// TwinCAT 3 PLC project MiniRobotPLC
// ProgramVersion: 3.1.4024.0
// libraries:
//   CL_GreenhouseObjectsLibrary, * (CleanGreensSA)
//   Tc2_MC2, * (Beckhoff Automation GmbH)
//   Tc2_Standard, * (Beckhoff Automation GmbH)
//   Tc2_System, * (Beckhoff Automation GmbH)
//   Tc3_Module, * (Beckhoff Automation GmbH)
// project tree:
//   DUTs/ E_RequAxle.TcDUT, E_StepAxle.TcDUT, MainStm.TcDUT, ST_AnalogLimits.TcDUT, ST_Analog_HWI.TcDUT, ST_Axle.TcDUT, ST_CardState_HWI.TcDUT, ST_DriverAX8206_HWI.TcDUT, ST_GHMI.TcDUT, ST_HMI.TcDUT, ST_IrrigationLine.TcDUT, ST_JogMotorControl.TcDUT, ST_MainCabinet_HWI.TcDUT, ST_MainCabinet_HWQ.TcDUT, ST_MainPwrPhases_HWI.TcDUT, ST_ManualCtrlBtn.TcDUT, ST_OverCurrProtection_HWI.TcDUT, ST_OverCurrProtection_HWQ.TcDUT, ST_PhaseInfo.TcDUT, ST_PhasesCommon.TcDUT, ST_PositioningLaser_HWI.TcDUT, ST_PwrSupplyAX8620_HWI.TcDUT, ST_RemoteControl_HWI.TcDUT, ST_RobotIdentification_HWI.TcDUT, ST_RobotLineBox_HWI.TcDUT, ST_RobotLineBox_HWQ.TcDUT, ST_Robot_Axes.TcDUT, ST_Robot_HWI.TcDUT, ST_Robot_HWQ.TcDUT, ST_SystemStatus.TcDUT, ST_SystemStatus_AR.TcDUT, ST_SystemStatus_ARP.TcDUT, ST_UPS_HWI.TcDUT
//   GVLs/ G.TcGVL, GI.TcGVL (excluded from build), GIQ_Robot01.TcGVL, GQ.TcGVL
//   / PlcTask.TcTTO
//   POUs/ MAIN.TcPOU
// real-time tasks:
//   TASK PlcTask: cycle T#10ms, priority 20, ADS port 350
// motion (NC):
//   TASK NC-Task 1 SAF: cycle T#2ms, priority 4, ADS port 501
//   TASK NC-Task 1 SVB: cycle T#10ms, priority 8, ADS port 511
//   AXIS Axis 1 (id 1)
//     OtherSettings: AllowMotionCmdToSlave=true
//     encoder EncType=19
//       EncPara: MaxCount=#xffffffff
//     drive DrvType=16
//       DrvPara: MaxCount=#xffffffff, DriveControlDWord=#x00000100
//         Analog: TorqueSetpointScale=10, ScaleFactorActTorque=0.1
//         TimeComp: TaskDelayCycles=1
//     controller CtrType=1
//       CtrPara: PriorControlFactor=1
//         Observer: BandWidth=20
//   AXIS Axis 2 (id 2)
//     OtherSettings: AllowMotionCmdToSlave=true
//     encoder EncType=19
//       EncPara: MaxCount=#xffffffff
//     drive DrvType=16
//       DrvPara: MaxCount=#xffffffff, DriveControlDWord=#x00000100
//         Analog: TorqueSetpointScale=10, ScaleFactorActTorque=0.1
//         TimeComp: TaskDelayCycles=1
//     controller CtrType=1
//       CtrPara: PriorControlFactor=1
//         Observer: BandWidth=20
//   AXIS Axis 3 (id 3)
//     OtherSettings: AllowMotionCmdToSlave=true
//     encoder EncType=19
//       EncPara: MaxCount=#xffffffff
//     drive DrvType=16
//       DrvPara: MaxCount=#xffffffff, DriveControlDWord=#x00000100
//         Analog: TorqueSetpointScale=10, ScaleFactorActTorque=0.1
//         TimeComp: TaskDelayCycles=1
//     controller CtrType=1
//       CtrPara: PriorControlFactor=1
//         Observer: BandWidth=20
//   AXIS Axis 4 (id 4)
//     OtherSettings: AllowMotionCmdToSlave=true
//     encoder EncType=19
//       EncPara: MaxCount=#xffffffff
//     drive DrvType=16
//       DrvPara: MaxCount=#xffffffff, DriveControlDWord=#x00000100
//         Analog: TorqueSetpointScale=10, ScaleFactorActTorque=0.1
//         TimeComp: TaskDelayCycles=1
//     controller CtrType=1
//       CtrPara: PriorControlFactor=1
//         Observer: BandWidth=20
//   AXIS CGSMini_Robot01AxisLine1Front (id 5)
//     OtherSettings: AllowMotionCmdToSlave=true
//     encoder EncType=1
//     drive DrvType=5
//       Analog: TorqueSetpointScale=10, ScaleFactorActTorque=0.1
//     controller CtrType=1
//       CtrPara: PriorControlFactor=1
//         Observer: BandWidth=20
//   AXIS CGSMini_Robot01AxisLine1Back (id 6)
//     OtherSettings: AllowMotionCmdToSlave=true
//     encoder EncType=1
//     drive DrvType=5
//       Analog: TorqueSetpointScale=10, ScaleFactorActTorque=0.1
//     controller CtrType=1
//       CtrPara: PriorControlFactor=1
//         Observer: BandWidth=20
//   AXIS CGSMini_Robot01AxisLine2Front (id 7)
//     OtherSettings: AllowMotionCmdToSlave=true
//     encoder EncType=1
//     drive DrvType=5
//       Analog: TorqueSetpointScale=10, ScaleFactorActTorque=0.1
//     controller CtrType=1
//       CtrPara: PriorControlFactor=1
//         Observer: BandWidth=20
//   AXIS CGSMini_Robot01AxisLine2Back (id 8)
//     OtherSettings: AllowMotionCmdToSlave=true
//     encoder EncType=1
//     drive DrvType=5
//       Analog: TorqueSetpointScale=10, ScaleFactorActTorque=0.1
//     controller CtrType=1
//       CtrPara: PriorControlFactor=1
//         Observer: BandWidth=20
// I/O:
//   DEVICE CGSMini_IRSMainPLCNoSafe, AmsNetId 5.93.147.0.3.1
//     CGSMini_RobotAllMainCab-EL1200
// variable links:
//   MiniRobotPLC Instance <-> CGSMini_IRSMainPLCNoSafe/CGSMini_RobotAllMainCab-EL1200/CGSMini_Robot01LineBoxAnaInN01-EL3202
//     PlcTask Inputs/GIQ_Robot01.stBoxIN/stAnaInN01_3202State/uiDataState <-> InfoData/State
//     PlcTask Inputs/GIQ_Robot01.stBoxIN/stAnaRTDLine1/bTError <-> RTD1/Status/Error
//     PlcTask Inputs/GIQ_Robot01.stBoxIN/stAnaRTDLine2/bTError <-> RTD2/Status/Error
//     PlcTask Inputs/GIQ_Robot01.stBoxIN/stAnaRTDLine1/bTLimit1 <-> RTD1/Status/Limit 1
//     PlcTask Inputs/GIQ_Robot01.stBoxIN/stAnaRTDLine1/bTLimit2 <-> RTD1/Status/Limit 2
//     PlcTask Inputs/GIQ_Robot01.stBoxIN/stAnaRTDLine2/bTLimit1 <-> RTD2/Status/Limit 1
//     PlcTask Inputs/GIQ_Robot01.stBoxIN/stAnaRTDLine2/bTLimit2 <-> RTD2/Status/Limit 2
//     PlcTask Inputs/GIQ_Robot01.stBoxIN/stAnaRTDLine1/bTOverRange <-> RTD1/Status/Overrange
//     PlcTask Inputs/GIQ_Robot01.stBoxIN/stAnaRTDLine2/bTOverRange <-> RTD2/Status/Overrange
//     PlcTask Inputs/GIQ_Robot01.stBoxIN/stAnaRTDLine1/bTUnderRange <-> RTD1/Status/Underrange
//     PlcTask Inputs/GIQ_Robot01.stBoxIN/stAnaRTDLine2/bTUnderRange <-> RTD2/Status/Underrange
//     PlcTask Inputs/GIQ_Robot01.stBoxIN/stAnaRTDLine1/siAnaRaw <-> RTD1/Value
//     PlcTask Inputs/GIQ_Robot01.stBoxIN/stAnaRTDLine2/siAnaRaw <-> RTD2/Value
//   MiniRobotPLC Instance <-> CGSMini_IRSMainPLCNoSafe/CGSMini_RobotAllMainCab-EL1200/CGSMini_Robot01LineBoxAnaInN02-EL3054
//     PlcTask Inputs/GIQ_Robot01.stBoxIN/stAnaFlowLine1/bTError <-> Flow1/Status/Error
//     PlcTask Inputs/GIQ_Robot01.stBoxIN/stAnaFlowLine2/bTError <-> Flow2/Status/Error
//     PlcTask Inputs/GIQ_Robot01.stBoxIN/stAnaFlowLine1/bTLimit1 <-> Flow1/Status/Limit 1
//     PlcTask Inputs/GIQ_Robot01.stBoxIN/stAnaFlowLine1/bTLimit2 <-> Flow1/Status/Limit 2
//     PlcTask Inputs/GIQ_Robot01.stBoxIN/stAnaFlowLine2/bTLimit1 <-> Flow2/Status/Limit 1
//     PlcTask Inputs/GIQ_Robot01.stBoxIN/stAnaFlowLine2/bTLimit2 <-> Flow2/Status/Limit 2
//     PlcTask Inputs/GIQ_Robot01.stBoxIN/stAnaFlowLine1/bTOverRange <-> Flow1/Status/Overrange
//     PlcTask Inputs/GIQ_Robot01.stBoxIN/stAnaFlowLine2/bTOverRange <-> Flow2/Status/Overrange
//     PlcTask Inputs/GIQ_Robot01.stBoxIN/stAnaFlowLine1/bTUnderRange <-> Flow1/Status/Underrange
//     PlcTask Inputs/GIQ_Robot01.stBoxIN/stAnaFlowLine2/bTUnderRange <-> Flow2/Status/Underrange
//     PlcTask Inputs/GIQ_Robot01.stBoxIN/stAnaFlowLine1/siAnaRaw <-> Flow1/Value
//     PlcTask Inputs/GIQ_Robot01.stBoxIN/stAnaFlowLine2/siAnaRaw <-> Flow2/Value
//     PlcTask Inputs/GIQ_Robot01.stBoxIN/stAnaInN02_3054State/uiDataState <-> InfoData/State
//     PlcTask Inputs/GIQ_Robot01.stBoxIN/stAnaPressure/bTError <-> Pressure1/Status/Error
//     PlcTask Inputs/GIQ_Robot01.stBoxIN/stAnaPressure/bTLimit1 <-> Pressure1/Status/Limit 1
//     PlcTask Inputs/GIQ_Robot01.stBoxIN/stAnaPressure/bTLimit2 <-> Pressure1/Status/Limit 2
//     PlcTask Inputs/GIQ_Robot01.stBoxIN/stAnaPressure/bTOverRange <-> Pressure1/Status/Overrange
//     PlcTask Inputs/GIQ_Robot01.stBoxIN/stAnaPressure/bTUnderRange <-> Pressure1/Status/Underrange
//     PlcTask Inputs/GIQ_Robot01.stBoxIN/stAnaPressure/siAnaRaw <-> Pressure1/Value
//   MiniRobotPLC Instance <-> CGSMini_IRSMainPLCNoSafe/CGSMini_RobotAllMainCab-EL1200/CGSMini_Robot01LineBoxAnaInN03-EL3202
//     PlcTask Inputs/GIQ_Robot01.stBoxIN/stAnaInN03_3202State/uiDataState <-> InfoData/State
//     PlcTask Inputs/GIQ_Robot01.stBoxIN/stAnaRTDExternal/bTError <-> RTDExternal/Status/Error
//     PlcTask Inputs/GIQ_Robot01.stBoxIN/stAnaRTDExternal/bTLimit1 <-> RTDExternal/Status/Limit 1
//     PlcTask Inputs/GIQ_Robot01.stBoxIN/stAnaRTDExternal/bTLimit2 <-> RTDExternal/Status/Limit 2
//     PlcTask Inputs/GIQ_Robot01.stBoxIN/stAnaRTDExternal/bTOverRange <-> RTDExternal/Status/Overrange
//     PlcTask Inputs/GIQ_Robot01.stBoxIN/stAnaRTDExternal/bTUnderRange <-> RTDExternal/Status/Underrange
//     PlcTask Inputs/GIQ_Robot01.stBoxIN/stAnaRTDExternal/siAnaRaw <-> RTDExternal/Value
//     PlcTask Inputs/GIQ_Robot01.stBoxIN/stAnaRTDInternal/bTError <-> RTDInternal/Status/Error
//     PlcTask Inputs/GIQ_Robot01.stBoxIN/stAnaRTDInternal/bTLimit1 <-> RTDInternal/Status/Limit 1
//     PlcTask Inputs/GIQ_Robot01.stBoxIN/stAnaRTDInternal/bTLimit2 <-> RTDInternal/Status/Limit 2
//     PlcTask Inputs/GIQ_Robot01.stBoxIN/stAnaRTDInternal/bTOverRange <-> RTDInternal/Status/Overrange
//     PlcTask Inputs/GIQ_Robot01.stBoxIN/stAnaRTDInternal/bTUnderRange <-> RTDInternal/Status/Underrange
//     PlcTask Inputs/GIQ_Robot01.stBoxIN/stAnaRTDInternal/siAnaRaw <-> RTDInternal/Value
//   MiniRobotPLC Instance <-> CGSMini_IRSMainPLCNoSafe/CGSMini_RobotAllMainCab-EL1200/CGSMini_Robot01LineBoxInN01-EL1008
//     PlcTask Inputs/GIQ_Robot01.stBoxIN/stInN01_1008State/uiDataState <-> InfoData/State
//     PlcTask Inputs/GIQ_Robot01.stBoxIN/stRemoteCtrl/BtnBackwardMan <-> Channel 2/BtnBackwardMan
//     PlcTask Inputs/GIQ_Robot01.stBoxIN/stRemoteCtrl/BtnForwardMan <-> Channel 1/BtnForwardMan
//     PlcTask Inputs/GIQ_Robot01.stBoxIN/stRemoteCtrl/BtnValveLine1Man <-> Channel 3/BtnValveLine1Man
//     PlcTask Inputs/GIQ_Robot01.stBoxIN/stRemoteCtrl/BtnValveLine2Man <-> Channel 4/BtnValveLine2Man
//     PlcTask Inputs/GIQ_Robot01.stBoxIN/stRobotID/bSelBit0 <-> Channel 5/SelLineBit0
//     PlcTask Inputs/GIQ_Robot01.stBoxIN/stRobotID/bSelBit1 <-> Channel 6/SelLineBit1
//     PlcTask Inputs/GIQ_Robot01.stBoxIN/stRobotID/bSelBit2 <-> Channel 7/SelLineBit2
//     PlcTask Inputs/GIQ_Robot01.stBoxIN/stRobotID/bSelBit3 <-> Channel 8/SelLineBit3
//   MiniRobotPLC Instance <-> CGSMini_IRSMainPLCNoSafe/CGSMini_RobotAllMainCab-EL1200/CGSMini_Robot01LineBoxOverCurrProt1-EL9222
//     PlcTask Inputs/GIQ_Robot01.stBoxIN/stOverCProt1_9222State/uiDataState <-> InfoData/State
//     PlcTask Inputs/GIQ_Robot01.stBoxIN/stOverCProt/bEnabled <-> OCP Inputs Channel 1/Status/Enabled
//     PlcTask Inputs/GIQ_Robot01.stBoxIN/stOverCProt/bError <-> OCP Inputs Channel 1/Status/Error
//   MiniRobotPLC Instance <-> CGSMini_IRSMainPLCNoSafe/CGSMini_RobotAllMainCab-EL1200/CGSMini_Robot01MainCabEtherCATBusEK1122/CGSMini_Robot01Laser-SickDL100
//     PlcTask Inputs/GIQ_Robot01.stIN/stLaserPos <-> Distance/Distance
//     PlcTask Inputs/GIQ_Robot01.stIN/stLaserPos_State/uiDataState <-> InfoData/State
//   MiniRobotPLC Instance <-> CGSMini_IRSMainPLCNoSafe/CGSMini_RobotAllMainCab-EL1200/CGSMini_Robot01MainCabEtherCATBusEK1122/CGSMini_Robot01OnboardAxisPwrSupply-AX8620
//     PlcTask Inputs/GIQ_Robot01.stIN/stPwrSupplyAX8620/bFanMalfunc <-> PSM Warning register/Warning/A4 Fan malfunction
//     PlcTask Inputs/GIQ_Robot01.stIN/stPwrSupplyAX8620/bOverTemp <-> PSM Warning register/Warning/A2 Device overtemperature
//     PlcTask Inputs/GIQ_Robot01.stIN/stPwrSupplyAX8620/bOverVoltage <-> PSM Warning register/Warning/A5 Mains overvoltage
//     PlcTask Inputs/GIQ_Robot01.stIN/stPwrSupplyAX8620/bUnderVoltage <-> PSM Warning register/Warning/A6 Mains undervoltage
//     PlcTask Inputs/GIQ_Robot01.stIN/stPwrSupplyAX8620/comState/bWcState <-> WcState/WcState
//     PlcTask Inputs/GIQ_Robot01.stIN/stPwrSupplyAX8620/comState/uiDataState <-> InfoData/State
//     PlcTask Inputs/GIQ_Robot01.stIN/stPwrSupplyAX8620/sdiDcInputShift <-> InfoData/DcInputShift
//     PlcTask Inputs/GIQ_Robot01.stIN/stPwrSupplyAX8620/sdiDcOutputShift <-> InfoData/DcOutputShift
//   MiniRobotPLC Instance <-> CGSMini_IRSMainPLCNoSafe/CGSMini_RobotAllMainCab-EL1200/CGSMini_Robot01MainCabEtherCATBusEK1122/CGSMini_Robot01OnboardAxisPwrSupply-AX8620/CGSMini_Robot01OnboardAxisDriverLine1-AX8206
//     PlcTask Inputs/GIQ_Robot01.stIN/stDriverLine1/comState <-> InfoData/State
//     PlcTask Inputs/GIQ_Robot01.stIN/stDriverLine1/rBackMotorTemp <-> Back/Ch A SyncServoMotor Inputs/Actual motor temperature
//     PlcTask Inputs/GIQ_Robot01.stIN/stDriverLine1/rBackMotorTorque <-> Back/Ch A TorqueControl Inputs/Ch A Torque/force actual value
//     PlcTask Inputs/GIQ_Robot01.stIN/stDriverLine1/rFrontMotorTemp <-> Front/Ch B SyncServoMotor Inputs/Actual motor temperature
//     PlcTask Inputs/GIQ_Robot01.stIN/stDriverLine1/rFrontMotorTorque <-> Front/Ch B TorqueControl Inputs/Ch B Torque/force actual value
//     PlcTask Inputs/GIQ_Robot01.stIN/stDriverLine1/sdiDcInputShift <-> InfoData/DcInputShift
//     PlcTask Inputs/GIQ_Robot01.stIN/stDriverLine1/sdiDcOutputShift <-> InfoData/DcOutputShift
//     PlcTask Inputs/GIQ_Robot01.stIN/stDriverLine1/siBackIGBTTemp <-> Back/Ch A AxisMain Inputs/IGBT temperature
//     PlcTask Inputs/GIQ_Robot01.stIN/stDriverLine1/siFrontIGBTTemp <-> Front/Ch B AxisMain Inputs/IGBT temperature
//     PlcTask Inputs/GIQ_Robot01.stIN/stDriverLine1/udBackMotorDIGIns <-> Back/Ch A AxisMain Inputs/Ch A Digital inputs
//     PlcTask Inputs/GIQ_Robot01.stIN/stDriverLine1/udFrontMotorDIGIns <-> Front/Ch B AxisMain Inputs/Ch B Digital inputs
//   MiniRobotPLC Instance <-> CGSMini_IRSMainPLCNoSafe/CGSMini_RobotAllMainCab-EL1200/CGSMini_Robot01MainCabEtherCATBusEK1122/CGSMini_Robot01OnboardAxisPwrSupply-AX8620/CGSMini_Robot01OnboardAxisDriverLine2-AX8206
//     PlcTask Inputs/GIQ_Robot01.stIN/stDriverLine2/comState <-> InfoData/State
//     PlcTask Inputs/GIQ_Robot01.stIN/stDriverLine2/rBackMotorTemp <-> Back/Ch A SyncServoMotor Inputs/Actual motor temperature
//     PlcTask Inputs/GIQ_Robot01.stIN/stDriverLine2/rBackMotorTorque <-> Back/Ch A TorqueControl Inputs/Ch A Torque/force actual value
//     PlcTask Inputs/GIQ_Robot01.stIN/stDriverLine2/rFrontMotorTemp <-> Front/Ch B SyncServoMotor Inputs/Actual motor temperature
//     PlcTask Inputs/GIQ_Robot01.stIN/stDriverLine2/rFrontMotorTorque <-> Front/Ch B TorqueControl Inputs/Ch B Torque/force actual value
//     PlcTask Inputs/GIQ_Robot01.stIN/stDriverLine2/sdiDcInputShift <-> InfoData/DcInputShift
//     PlcTask Inputs/GIQ_Robot01.stIN/stDriverLine2/sdiDcOutputShift <-> InfoData/DcOutputShift
//     PlcTask Inputs/GIQ_Robot01.stIN/stDriverLine2/siBackIGBTTemp <-> Back/Ch A AxisMain Inputs/IGBT temperature
//     PlcTask Inputs/GIQ_Robot01.stIN/stDriverLine2/siFrontIGBTTemp <-> Front/Ch B AxisMain Inputs/IGBT temperature
//     PlcTask Inputs/GIQ_Robot01.stIN/stDriverLine2/udBackMotorDIGIns <-> Back/Ch A AxisMain Inputs/Ch A Digital inputs
//     PlcTask Inputs/GIQ_Robot01.stIN/stDriverLine2/udFrontMotorDIGIns <-> Front/Ch B AxisMain Inputs/Ch B Digital inputs
//   MiniRobotPLC Instance <-> CGSMini_IRSMainPLCNoSafe/CGSMini_RobotAllMainCab-EL1200/CGSMini_Robot01MainCabEtherCATBusEK1122/CGSMini_Robot01OnboardBox-EK1100
//     PlcTask Inputs/GIQ_Robot01.stIN/stOnboardBox_1100State/uiDataState <-> InfoData/State
//   MiniRobotPLC Instance <-> CGSMini_IRSMainPLCNoSafe/CGSMini_RobotAllMainCab-EL1200/CGSMini_Robot01MainCabEtherCATBusEK1122/CGSMini_Robot01OnboardBox-EK1100/CGSMini_Robot01OnBoardBoxAnaInN04-EL3054
//     PlcTask Inputs/GIQ_Robot01.stIN/stAnaInN04_3054State/uiDataState <-> InfoData/State
//     PlcTask Inputs/GIQ_Robot01.stIN/stAnaOnboardSpare1/bTError <-> Spare1/Status/Error
//     PlcTask Inputs/GIQ_Robot01.stIN/stAnaOnboardSpare1/bTLimit1 <-> Spare1/Status/Limit 1
//     PlcTask Inputs/GIQ_Robot01.stIN/stAnaOnboardSpare1/bTLimit2 <-> Spare1/Status/Limit 2
//     PlcTask Inputs/GIQ_Robot01.stIN/stAnaOnboardSpare1/bTOverRange <-> Spare1/Status/Overrange
//     PlcTask Inputs/GIQ_Robot01.stIN/stAnaOnboardSpare1/bTUnderRange <-> Spare1/Status/Underrange
//     PlcTask Inputs/GIQ_Robot01.stIN/stAnaOnboardSpare1/siAnaRaw <-> Spare1/Value
//   MiniRobotPLC Instance <-> CGSMini_IRSMainPLCNoSafe/CGSMini_RobotAllMainCab-EL1200/CGSMini_Robot01MainCabEtherCATBusEK1122/CGSMini_Robot01OnboardBox-EK1100/CGSMini_Robot01OnBoardBoxOutN01-EL2008
//     PlcTask Inputs/GIQ_Robot01.stIN/stOutN01_2008State/uiDataState <-> InfoData/State
//     PlcTask Outputs/G.outTest14 <-> Channel 8/Output
//     PlcTask Outputs/GIQ_Robot01.stOUT/FlushFloor <-> Channel 1/FlushFloor
//     PlcTask Outputs/GIQ_Robot01.stOUT/IrrigLine1 <-> Channel 3/IrrigLine1
//     PlcTask Outputs/GIQ_Robot01.stOUT/IrrigLine2 <-> Channel 4/IrrigLine2
//   MiniRobotPLC Instance <-> CGSMini_IRSMainPLCNoSafe/CGSMini_RobotAllMainCab-EL1200/CGSMini_RobotAllMainCabOutN01-EL2008
//     PlcTask Outputs/GQ.stMainCabinet/bEmgyBtnRedLight <-> Channel 3/EmgyBtnRedLight
//     PlcTask Outputs/GQ.stMainCabinet/bEmgyBtnWhiteLight <-> Channel 2/EmgyBtnWhiteLight
//     PlcTask Outputs/GQ.stMainCabinet/stStackLight/bBlue <-> Channel 4/blue
//     PlcTask Outputs/GQ.stMainCabinet/stStackLight/bBuzzer <-> Channel 8/buzzer
//     PlcTask Outputs/GQ.stMainCabinet/stStackLight/bGreen <-> Channel 5/green
//     PlcTask Outputs/GQ.stMainCabinet/stStackLight/bOrange <-> Channel 6/orange
//     PlcTask Outputs/GQ.stMainCabinet/stStackLight/bRed <-> Channel 7/red
//   MiniRobotPLC Instance <-> NC-Task 1 SAF/Axes/CGSMini_Robot01AxisLine1Back
//     PlcTask Inputs/GIQ_Robot01.stAxes.Line1Back.NcToPlc <-> Outputs/ToPlc
//     PlcTask Outputs/GIQ_Robot01.stAxes.Line1Back.PlcToNc <-> Inputs/FromPlc
//   MiniRobotPLC Instance <-> NC-Task 1 SAF/Axes/CGSMini_Robot01AxisLine1Front
//     PlcTask Inputs/GIQ_Robot01.stAxes.Line1Front.NcToPlc <-> Outputs/ToPlc
//     PlcTask Outputs/GIQ_Robot01.stAxes.Line1Front.PlcToNc <-> Inputs/FromPlc
//   MiniRobotPLC Instance <-> NC-Task 1 SAF/Axes/CGSMini_Robot01AxisLine2Back
//     PlcTask Inputs/GIQ_Robot01.stAxes.Line2Back.NcToPlc <-> Outputs/ToPlc
//     PlcTask Outputs/GIQ_Robot01.stAxes.Line2Back.PlcToNc <-> Inputs/FromPlc
//   MiniRobotPLC Instance <-> NC-Task 1 SAF/Axes/CGSMini_Robot01AxisLine2Front
//     PlcTask Inputs/GIQ_Robot01.stAxes.Line2Front.NcToPlc <-> Outputs/ToPlc
//     PlcTask Outputs/GIQ_Robot01.stAxes.Line2Front.PlcToNc <-> Inputs/FromPlc

CONFIGURATION MiniRobotPLC
    RESOURCE PLC ON TwinCAT3
        TASK PlcTask(INTERVAL := T#10ms, PRIORITY := 20);
        PROGRAM MAIN WITH PlcTask : MAIN;
    END_RESOURCE
END_CONFIGURATION

// ---- DUTs/E_RequAxle.TcDUT
{attribute 'qualified_only'}
{attribute 'strict'}
TYPE E_RequAxle :
(
  NoRequ := 0,
  PowerOn := 1,
  PowerOff := 2,
  Reset := 3,
  Jog := 4,
  Error := 254,
  Idle := 255
);
END_TYPE

// ---- DUTs/E_StepAxle.TcDUT
{attribute 'qualified_only'}
{attribute 'strict'}
TYPE E_StepAxle :
(
	//Idle	        := 0,
  Init          := 1,
  
	// STEPS ABSOLUTE
 	MoveAbs		    := 11,
	EndMoveAbs    := 12,
  
	// STEPS STOP
  InitStop      := 50,
	Stopping		  := 51,
  EndStopping   := 52,
	
	// STEPS HOMING
  InitHoming    := 60,
	Homing			  := 61,
  EndHoming     := 62,
  InitAbortHoming := 63,
  AbortHoming   := 64,
  InitRetryHoming := 65,
  RetryHoming     := 66,
	
	// STEPS Reset
  ResetTimeout := 70,
	Resetting	:= 71,
  ResetEnd := 72,
  
  // step jogs
  JogMoveFW := 80,
  JogMoveBW := 81,
  JogStop := 82,
  JogEnd := 83
);
END_TYPE

// ---- DUTs/MainStm.TcDUT
{attribute 'qualified_only'}
{attribute 'strict'}
TYPE MainStm :
(
	ModuleDatabaseInit := 0,
  ModuleDatabaseLoad,
  ErrorDatabaseInit,
	LoadSQLDB,
  Init,
	//WaitInitWebVISUTask,
	LoadModuleDB,
	InitWebVISUTask,
	IRSystemExec,//GreenhouseExec,
	PowerFailure,
	WaitPowerDown,
	ReqShutdown,
  ReqRestart,
  FailedLoadSQL,
  FailedInitObjects,
	End
);
END_TYPE

// ---- DUTs/ST_AnalogLimits.TcDUT
TYPE ST_AnalogLimits :
STRUCT
  lrAroundZero        : LREAL; //to check if the value is around zero
	lrRawLowerLimit		  : LREAL; // Lower limit for raw data
	lrRawUpperLimit		  : LREAL; // Upper limit for raw data
	lrScaleLowerLimit	  : LREAL; // Lower limit of scaled measurement
	lrScaleUpperLimit	  : LREAL; // Upper limit of scaled measurement
  bForceZero          : BOOL;
END_STRUCT
END_TYPE

// ---- DUTs/ST_Analog_HWI.TcDUT
TYPE ST_Analog_HWI :
STRUCT
  bTUnderRange      : BOOL;
  bTOverRange       : BOOL;
  bTLimit1          : BOOL;
  bTLimit2          : BOOL;
  bTError           : BOOL;
  siAnaRaw          : INT;  
END_STRUCT
END_TYPE

// ---- DUTs/ST_Axle.TcDUT
//Add Library Tc2_MC2
TYPE ST_Axle:
STRUCT
	stAxisRef						      : POINTER TO AXIS_REF;//axis reference linked to I/O
	fbPower						        : MC_Power;//Axis function - Power
	fbReset						        : MC_Reset;//Axis function - Reset
	fbSetPosition					    : MC_SetPosition;//Axis function - Set Position
	fbStop							      : MC_Stop;//stop
	fbHalt							      : MC_Halt;//Halt
	fbHome							      : MC_Home;//Home
	fbMoveJog							    : MC_Jog;//Jog
  fbReadStatus              : MC_ReadStatus;
	fbMoveAbsolute1				    : MC_MoveAbsolute;//	MC_MoveAbsolute1
  fbMoveAbsoluteWheelCheck  : MC_MoveAbsolute;// Add CustomAutomation 07.03.2023: Check du diamètre des roues 
  fbMoveAbsoluteCorrection  : MC_MoveAbsolute;// Add CustomAutomation 07.03.2023: Correction fin de parcours
 	fbMoveRelative					  : MC_MoveRelative;//Move Relative
	fbMoveVelocity					  : MC_MoveVelocity;//Move Velocity
	fbReadAxisError				    : MC_ReadAxisError;//Status and parameter - Read Axis Error
	fbReadActualPosition			: MC_ReadActualPosition;//Status and parameter - Read Actual Position
	fbReadActualVelocity			: MC_ReadActualVelocity;//Status and parameter - Read Actual Velocity
	fbGearInDyn					      : MC_GearInDyn;//Axis coupling - GearInDyn
	fbGearOut						      : MC_GearOut;//Axis coupling - GearOut
	fbPosCorrectionLimiter    : MC_PositionCorrectionLimiter;//Special extensions - Position Correction Limiter
	
	bGearOutDone					    : BOOL;
	bGearInDynDone					  : BOOL;
	bStopDone						      : BOOL;
END_STRUCT
END_TYPE

// ---- DUTs/ST_CardState_HWI.TcDUT
TYPE ST_CardState_HWI :
STRUCT
  uiDataState   : UINT;
  bWcState      : BOOL := FALSE;
END_STRUCT
END_TYPE

// ---- DUTs/ST_DriverAX8206_HWI.TcDUT

TYPE ST_DriverAX8206_HWI :
STRUCT
  comState          : ST_CardState_HWI;
  sdiDcOutputShift  : DINT;
  sdiDcInputShift   : DINT;

  siFrontIGBTTemp   : INT;//ChB
  siBackIGBTTemp    : INT;//ChA
  
  rFrontMotorTemp  : REAL;//ChB
  rBackMotorTemp   : REAL;//ChA
  
  rFrontMotorTorque : REAL;//ChB
  rBackMotorTorque  : REAL;//ChA
  
  udFrontMotorDIGIns: UDINT;//ChB
  udBackMotorDIGIns: UDINT;//ChA
END_STRUCT
END_TYPE

// ---- DUTs/ST_GHMI.TcDUT
TYPE ST_GHMI :
STRUCT
  bStartButton      		  : BOOL;
  bStopButton       		  : BOOL;
  bResetButton      		  : BOOL;
  bAbortButton      		  : BOOL;
  bClearButton      		  : BOOL;
  nIndexFrame       		  : INT := 0;
  nIndexFrameAdmin        : INT := 0;
  nIndexFrameHome   		  : INT := 0;
  bPopUpModulPresent		  : BOOL;
  bPopUpHoming      		  : BOOL;
  bPopUpExtractorAborted  : BOOL;
	bPopUpInsertModulesLine	: BOOL;
  bRestart          		  : BOOL;
  bShutdown          		  : BOOL;
	sBtnAdmin								: STRING(32);
END_STRUCT
END_TYPE

// ---- DUTs/ST_HMI.TcDUT
TYPE ST_HMI :
STRUCT
  nIrrLineSel  : UINT := 1;//at leat 1 robot line
END_STRUCT
END_TYPE

// ---- DUTs/ST_IrrigationLine.TcDUT
TYPE ST_IrrigationLine :
STRUCT
  stRobotLineBoxHWI   : POINTER TO ST_RobotLineBox_HWI;
  stRobotLineBoxHWQ   : POINTER TO ST_RobotLineBox_HWQ;
  stRobotHWI	        : POINTER TO ST_Robot_HWI;
  stRobotHWQ	        : POINTER TO ST_Robot_HWQ;
  stRobotAxes	        : POINTER TO ST_Robot_Axes;
END_STRUCT
END_TYPE

// ---- DUTs/ST_JogMotorControl.TcDUT
TYPE ST_JogMotorControl :
STRUCT
  bMoveFW   : BOOL := false;
  bMoveBW   : BOOL := false;
END_STRUCT
END_TYPE

// ---- DUTs/ST_MainCabinet_HWI.TcDUT
TYPE ST_MainCabinet_HWI :
STRUCT		
    //State
    stInN01_1008State       : ST_CardState_HWI;
    stOutN01_2008State      : ST_CardState_HWI; 
    stLicense_6070State     : ST_CardState_HWI; 
    stAnaInN01_3443         : ST_CardState_HWI; //CGSMini_RobotAllMainCabAnaInN01-EL3443
    
    //EK1122 ethercat State    
    stMainEK1122State       : ST_CardState_HWI;
    
		//inputs
		bKeyRestart			 	 			: BOOL;  
		bEmgyBtnCntct1					: BOOL; 
		bEmgyBtnCntct2	   			: BOOL;  
		bOverTemp45C			 			: BOOL := FALSE;  
    bPLCCircuitBreakerOpen  : BOOL := FALSE;   
    
    stUPS                   : ST_UPS_HWI;
    stPwrInfo               : ST_MainPwrPhases_HWI;
END_STRUCT
END_TYPE

// ---- DUTs/ST_MainCabinet_HWQ.TcDUT
TYPE ST_MainCabinet_HWQ :
STRUCT
  //outputs
  bEmgyBtnWhiteLight  	: BOOL;  
  bEmgyBtnRedLight  		: BOOL; 
  
  stStackLight          : ST_StackLight_HWQ;
END_STRUCT
END_TYPE

// ---- DUTs/ST_MainPwrPhases_HWI.TcDUT
TYPE ST_MainPwrPhases_HWI :
STRUCT
  L1 : ST_PhaseInfo;
  L2 : ST_PhaseInfo;
  L3 : ST_PhaseInfo;
  Tot : ST_PhasesCommon;
END_STRUCT
END_TYPE

// ---- DUTs/ST_ManualCtrlBtn.TcDUT
TYPE ST_ManualCtrlBtn :
STRUCT
  bMoveBackwardBtn        : BOOL := FALSE;
  bMoveForwardBtn         : BOOL := FALSE;
  bVlvLine1Btn            : BOOL := FALSE;
  bVlvLine2Btn            : BOOL := FALSE;
  
  bMoveBackwardBtnPress   : BOOL := FALSE;
  bMoveForwardBtnPress    : BOOL := FALSE;
  bVlvLine1BtnPress       : BOOL := FALSE;
  bVlvLine2BtnPress       : BOOL := FALSE;
END_STRUCT
END_TYPE

// ---- DUTs/ST_OverCurrProtection_HWI.TcDUT
TYPE ST_OverCurrProtection_HWI :
STRUCT
  bEnabled  : BOOL;
  bError    : BOOL;
END_STRUCT
END_TYPE

// ---- DUTs/ST_OverCurrProtection_HWQ.TcDUT
TYPE ST_OverCurrProtection_HWQ :
STRUCT
  bCtrlResetCh1   : BOOL;
  bCtrlSwitchCh1  : BOOL;
  bCtrlResetCh2   : BOOL;
  bCtrlSwitchCh2  : BOOL;
END_STRUCT
END_TYPE

// ---- DUTs/ST_PhaseInfo.TcDUT
TYPE ST_PhaseInfo :
STRUCT
  Voltage : REAL;
  Current : REAL;
END_STRUCT
END_TYPE

// ---- DUTs/ST_PhasesCommon.TcDUT
TYPE ST_PhasesCommon :
STRUCT
  L1_L2_V : REAL;
END_STRUCT
END_TYPE

// ---- DUTs/ST_PositioningLaser_HWI.TcDUT
TYPE ST_PositioningLaser_HWI :
STRUCT
  udiDistanceRaw          : UDINT;  
END_STRUCT
END_TYPE

// ---- DUTs/ST_PwrSupplyAX8620_HWI.TcDUT
TYPE ST_PwrSupplyAX8620_HWI :
STRUCT
  comState          : ST_CardState_HWI;
  sdiDcOutputShift  : DINT;
  sdiDcInputShift   : DINT;

  bOverTemp         : BOOL;
  bFanMalfunc       : BOOL;
  bUnderVoltage     : BOOL; // Power supply undervoltage
  bOverVoltage      : BOOL; // Power supply overvoltage
END_STRUCT
END_TYPE

// ---- DUTs/ST_RemoteControl_HWI.TcDUT
TYPE ST_RemoteControl_HWI:
STRUCT
  BtnForwardMan     : BOOL := false;
  BtnBackwardMan    : BOOL := false;
  BtnValveLine1Man  : BOOL := false;
  BtnValveLine2Man  : BOOL := false;
END_STRUCT
END_TYPE

// ---- DUTs/ST_RobotIdentification_HWI.TcDUT
TYPE ST_RobotIdentification_HWI :
STRUCT
    bSelBit0                : BOOL;
    bSelBit1                : BOOL;
    bSelBit2                : BOOL;
    bSelBit3                : BOOL;
END_STRUCT
END_TYPE

// ---- DUTs/ST_RobotLineBox_HWI.TcDUT
TYPE ST_RobotLineBox_HWI :
STRUCT
  stInN01_1008State       : ST_CardState_HWI;//CGSMini_Robot01LineBoxInN01-EL1008
  stAnaInN01_3202State    : ST_CardState_HWI;//CGSMini_Robot01LineBoxAnaInN01-EL3202
  stAnaInN02_3054State    : ST_CardState_HWI;//CGSMini_Robot01LineBoxAnaInN02-EL3054
  stAnaInN03_3202State    : ST_CardState_HWI;//CGSMini_Robot01LineBoxAnaInN03-EL3202
  stOverCProt1_9222State  : ST_CardState_HWI;//CGSMini_Robot01LineBoxOverCurrProt1-EL9222
  stLineBox_1100State     : ST_CardState_HWI;//CGSMini_Robot01LineBoxBox-EK1100 not yet available useful in case of only one PLC for all robots line
  stSafety_1918State      : ST_CardState_HWI;//CGSMini_Robot01LineBoxSafeInN01-EL1918
 
  stRobotID               : ST_RobotIdentification_HWI;//CGSMini_Robot01LineBoxInN01-EL1008
  stRemoteCtrl            : ST_RemoteControl_HWI;//CGSMini_Robot01LineBoxInN01-EL1008
  stOverCProt             : ST_OverCurrProtection_HWI;//CGSMini_Robot01LineBoxOverCurrProt1-EL9222
  stAnaRTDLine1           : ST_Analog_HWI;//CGSMini_Robot01LineBoxAnaInN01-EL3202 RTD1
  stAnaRTDLine2           : ST_Analog_HWI;//CGSMini_Robot01LineBoxAnaInN01-EL3202 RTD2
	stAnaFlowLine1          : ST_Analog_HWI;//CGSMini_Robot01LineBoxAnaInN02-EL3054 
  stAnaFlowLine2          : ST_Analog_HWI;//CGSMini_Robot01LineBoxAnaInN02-EL3054 
  stAnaPressure           : ST_Analog_HWI;//CGSMini_Robot01LineBoxAnaInN02-EL3054
  stAnaRTDInternal        : ST_Analog_HWI;//CGSMini_Robot01LineBoxAnaInN03-EL3202 RTDInternal
  stAnaRTDExternal        : ST_Analog_HWI;//CGSMini_Robot01LineBoxAnaInN03-EL3202 RTDExternal
END_STRUCT
END_TYPE

// ---- DUTs/ST_RobotLineBox_HWQ.TcDUT
TYPE ST_RobotLineBox_HWQ :
STRUCT
  stOverCProt : ST_OverCurrProtection_HWQ;//CGSMini_Robot01LineBoxOverCurrProt1-EL9222
END_STRUCT
END_TYPE

// ---- DUTs/ST_Robot_Axes.TcDUT
TYPE ST_Robot_Axes :
STRUCT
  Line1Front    : AXIS_REF;//Axis4-Line1-Left Front (ChB) - second Drive in I/O Tree
  Line1Back     : AXIS_REF;//Axis3-Line1-Left Back (ChA) - second Drive in I/O Tree
  Line2Front    : AXIS_REF;//Axis2-Line2-Right Front (ChB) - first Drive in I/O Tree
  Line2Back     : AXIS_REF;//Axis1-Line2-Right Back (ChA)- first Drive in I/O Tree
END_STRUCT
END_TYPE

(*
Old Robot HW Drivers assign table
ChA -> Front
ChB -> Back
Axe1-LA-Left Front-GVL_Intern.arAxe[1] - Drive 8 (AX8206-0200-0104) # 'Ch A'
Axe2-LB-Left Back-GVL_Intern.arAxe[2] - Drive 8 (AX8206-0200-0104) # 'Ch B'
Axe3-RA-Right Front-GVL_Intern.arAxe[3] - Drive 9 (AX8206-0200-0104) # 'Ch A'
Axe4-RB-Right Back-GVL_Intern.arAxe[4] - Drive 9 (AX8206-0200-0104) # 'Ch B'
*)

// ---- DUTs/ST_Robot_HWI.TcDUT
TYPE ST_Robot_HWI :
STRUCT
  stAnaInN04_3054State    : ST_CardState_HWI;//CGSMini_Robot01OnBoardBoxAnaInN04-EL3054
  stOnboardBox_1100State  : ST_CardState_HWI;//CGSMini_Robot01OnboardBox-EK1100
  stLaserPos_State        : ST_CardState_HWI;//CGSMini_Robot01Laser-SickDL100
  stOutN01_2008State      : ST_CardState_HWI;//CGSMini_Robot01OnBoardBoxOutN01-EL2008
  
  stLaserPos              : ST_PositioningLaser_HWI;//CGSMini_Robot01Laser-SickDL100
  stAnaOnboardSpare1      : ST_Analog_HWI;//CGSMini_Robot01OnBoardBoxAnaInN04-EL3054
  stPwrSupplyAX8620       : ST_PwrSupplyAX8620_HWI;//CGSMini_Robot01OnboardAxisAlim-AX8620
  stDriverLine1           : ST_DriverAX8206_HWI;
  stDriverLine2           : ST_DriverAX8206_HWI;
 END_STRUCT
END_TYPE

// ---- DUTs/ST_Robot_HWQ.TcDUT
TYPE ST_Robot_HWQ :
STRUCT
  	//OutN01
		FlushFloor  	          : BOOL;  
		IrrigLine1  		        : BOOL;
    IrrigLine2    	        : BOOL; 
END_STRUCT
END_TYPE

// ---- DUTs/ST_SystemStatus.TcDUT
TYPE ST_SystemStatus :
STRUCT
  nRequestModeMachine      : E_ModeMachine := E_ModeMachine.Startup;
  nModeMachine             : E_ModeMachine := E_ModeMachine.Startup;
  nStateMachine            : E_StateMachine := E_StateMachine.cIdle;
END_STRUCT
END_TYPE

// ---- DUTs/ST_SystemStatus_AR.TcDUT
TYPE 
  ST_SystemStatus_AR : ARRAY [0..C.uiNumRobotForHMI_C] OF ST_SystemStatus;
END_TYPE

// ---- DUTs/ST_SystemStatus_ARP.TcDUT
TYPE
  ST_SystemStatus_ARP : POINTER TO ARRAY [0..C.uiNumRobotForHMI_C] OF ST_SystemStatus;
END_TYPE

// ---- DUTs/ST_UPS_HWI.TcDUT
TYPE ST_UPS_HWI :
STRUCT
  bPowerReady	      	: BOOL;
  bPowerFail		      : BOOL;	
END_STRUCT
END_TYPE

// ---- GVLs/G.TcGVL
{attribute 'qualified_only'}
VAR_GLOBAL
  //{attribute 'TcLinkTo' := 'TIIB[Term4EL2008]^Channel 1^Output'}
  //outTest4 AT %Q* : BOOL;

  //{attribute 'TcLinkTo' := 'TIIB[Term14EL2008]^Channel 8^Output;'}
  //outTest14 AT %Q* : BOOL;

  {attribute 'TcLinkTo' := 'TIIB[CGSMini_Robot01OnBoardBoxOutN01-EL2008]^Channel 8^Output;'}
  outTest14 AT %Q* : BOOL;
END_VAR

// ---- GVLs/GI.TcGVL
{attribute 'qualified_only'}
{IF defined (debugCompile)}
 //contains ONLY global variable to access hardware input debugCompile mode
{info '---------------simulation input global variables used; DEBUG defined---------------'}
VAR_GLOBAL	
  stMainCabinet : ST_MainCabinet_HWI;
END_VAR    
{END_IF}

VAR_GLOBAL
  {attribute 'TcLinkTo':='outFloor := TIIB[Term 14 (EL2008)]^Channel 1^Output;}
  outFloor AT %Q*:BOOL;

  {info '---------------Hardware inputs used; CGSMiniRobot defined---------------'}		
  {attribute 'TcLinkTo':='.bKeyRestart                := TIIB[CGSMini_RobotAllMainCabInN01-EL1008]^Channel 1^KeyRestart;
                      .bEmgyBtnCntct1                 := TIIB[CGSMini_RobotAllMainCabInN01-EL1008]^Channel 2^EmgyBtnCntct1;
                      .bEmgyBtnCntct2                 := TIIB[CGSMini_RobotAllMainCabInN01-EL1008]^Channel 3^EmgyBtnCntct2;
                      .bOverTemp45C                   := TIIB[CGSMini_RobotAllMainCabInN01-EL1008]^Channel 5^OverTemp45C;
                      .bPLCCircuitBreakerOpen         := TIIB[CGSMini_RobotAllMainCabInN01-EL1008]^Channel 6^PLCCircuitBreakerOpen;
                      
                      .stUPS.bPowerReady              := TIIB[CGSMini_RobotAllMainCabInN01-EL1008]^Channel 8^UPSPowerReady;
                      .stUPS.bPowerFail               := TIIB[CGSMini_RobotAllMainCabInN01-EL1008]^Channel 7^UPSPowerFail;
                      
                      .stPwrInfo.L1.Voltage           := TIIB[CGSMini_RobotAllMainCabAnaInN01-EL3443]^L1 Basic^Voltage;
                      .stPwrInfo.L1.Current           := TIIB[CGSMini_RobotAllMainCabAnaInN01-EL3443]^L1 Basic^Current;
                      .stPwrInfo.Tot.L1_L2_V          := TIIB[CGSMini_RobotAllMainCabAnaInN01-EL3443]^Total L-L Voltage^L1-L2 Voltage;
                   
                      .stMainEK1122State.uiDataState  := TIIB[CGSMini_Robot01MainCabEtherCATBusEK1122]^InfoData^State;
                      
                      .stInN01_1008State.uiDataState  := TIIB[CGSMini_RobotAllMainCabInN01-EL1008]^InfoData^State;
                      .stInN01_1008State.bWcState     := TIIB[CGSMini_RobotAllMainCabInN01-EL1008]^WcState^WcState;
                      
                      .stAnaInN01_3443.uiDataState    := TIIB[CGSMini_RobotAllMainCabAnaInN01-EL3443]^InfoData^State;
                      .stAnaInN01_3443.bWcState       := TIIB[CGSMini_RobotAllMainCabAnaInN01-EL3443]^WcState^WcState;

                      .stOutN01_2008State.uiDataState := TIIB[CGSMini_RobotAllMainCabOutN01-EL2008]^InfoData^State;
                      .stOutN01_2008State.bWcState    := TIIB[CGSMini_RobotAllMainCabOutN01-EL2008]^WcState^WcState;

                      .stLicense_6070State.uiDataState := TIIB[CGSMini_RobotAllLicenses-EL6070]^InfoData^State;'}
  stMainCabinet AT %I* :ST_MainCabinet_HWI;	
END_VAR

// ---- GVLs/GIQ_Robot01.TcGVL
{attribute 'qualified_only'}

{IF defined (debugCompile)}
VAR_GLOBAL
	stIN	    : ST_Robot_HWI;	
  stBoxIN   : ST_RobotLineBox_HWI;
	stOUT     : ST_Robot_HWQ;
  stBoxOUT  : ST_RobotLineBox_HWQ;
  stAxes    : ST_Robot_Axes;
END_VAR
{END_IF}

VAR_GLOBAL
{attribute 'TcLinkTo':='.stInN01_1008State.uiDataState      := TIIB[CGSMini_Robot01LineBoxInN01-EL1008]^InfoData^State;
                        .stInN01_1008State.bWCState         := TIIB[CGSMini_Robot01LineBoxInN01-EL1008]^WcState^WcState;  
                        .stAnaInN01_3202State.uiDataState   := TIIB[CGSMini_Robot01LineBoxAnaInN01-EL3202]^InfoData^State;
                        .stAnaInN01_3202State.bWCState      := TIIB[CGSMini_Robot01LineBoxAnaInN01-EL3202]^WcState^WcState; 
                        .stAnaInN02_3054State.uiDataState   := TIIB[CGSMini_Robot01LineBoxAnaInN02-EL3054]^InfoData^State;
                        .stAnaInN02_3054State.bWCState      := TIIB[CGSMini_Robot01LineBoxAnaInN02-EL3054]^WcState^WcState; 
                        .stAnaInN03_3202State.uiDataState   := TIIB[CGSMini_Robot01LineBoxAnaInN03-EL3202]^InfoData^State;
                        .stAnaInN03_3202State.bWCState      := TIIB[CGSMini_Robot01LineBoxAnaInN03-EL3202]^WcState^WcState; 
                        .stOverCProt1_9222State.uiDataState := TIIB[CGSMini_Robot01LineBoxOverCurrProt1-EL9222]^InfoData^State;
                        .stOverCProt1_9222State.bWCState    := TIIB[CGSMini_Robot01LineBoxOverCurrProt1-EL9222]^WcState^WcState;                     
 
                        .stSafety_1918State.uiDataState     := TIIB[CGSMini_Robot01LineBoxSafeInN01-EL1918]^InfoData^State;
                        .stSafety_1918State.bWcState        := TIIB[CGSMini_Robot01LineBoxSafeInN01-EL1918]^WcState^WcState;

                        .stRemoteCtrl.BtnForwardMan         := TIIB[CGSMini_Robot01LineBoxInN01-EL1008]^Channel 1^BtnForwardMan;
                        .stRemoteCtrl.BtnBackwardMan        := TIIB[CGSMini_Robot01LineBoxInN01-EL1008]^Channel 2^BtnBackwardMan;
                        .stRemoteCtrl.BtnValveLine1Man      := TIIB[CGSMini_Robot01LineBoxInN01-EL1008]^Channel 3^BtnValveLine1Man;
                        .stRemoteCtrl.BtnValveLine2Man      := TIIB[CGSMini_Robot01LineBoxInN01-EL1008]^Channel 4^BtnValveLine2Man;
                       
                        .stRobotID.bSelBit0                 := TIIB[CGSMini_Robot01LineBoxInN01-EL1008]^Channel 5^SelLineBit0;
                        .stRobotID.bSelBit1                 := TIIB[CGSMini_Robot01LineBoxInN01-EL1008]^Channel 6^SelLineBit1;
                        .stRobotID.bSelBit2                 := TIIB[CGSMini_Robot01LineBoxInN01-EL1008]^Channel 7^SelLineBit2;
                        .stRobotID.bSelBit3                 := TIIB[CGSMini_Robot01LineBoxInN01-EL1008]^Channel 8^SelLineBit3;

                        .stAnaRTDLine1.bTUnderRange         := TIIB[CGSMini_Robot01LineBoxAnaInN01-EL3202]^RTD1^Status^Underrange;
                        .stAnaRTDLine1.bTOverRange          := TIIB[CGSMini_Robot01LineBoxAnaInN01-EL3202]^RTD1^Status^Overrange;
                        .stAnaRTDLine1.bTLimit1             := TIIB[CGSMini_Robot01LineBoxAnaInN01-EL3202]^RTD1^Status^Limit 1;
                        .stAnaRTDLine1.bTLimit2             := TIIB[CGSMini_Robot01LineBoxAnaInN01-EL3202]^RTD1^Status^Limit 2;
                        .stAnaRTDLine1.bTError              := TIIB[CGSMini_Robot01LineBoxAnaInN01-EL3202]^RTD1^Status^Error;
                        .stAnaRTDLine1.siAnaRaw             := TIIB[CGSMini_Robot01LineBoxAnaInN01-EL3202]^RTD1^Value;
 
                        .stAnaRTDLine2.bTUnderRange         := TIIB[CGSMini_Robot01LineBoxAnaInN01-EL3202]^RTD2^Status^Underrange;
                        .stAnaRTDLine2.bTOverRange          := TIIB[CGSMini_Robot01LineBoxAnaInN01-EL3202]^RTD2^Status^Overrange;
                        .stAnaRTDLine2.bTLimit1             := TIIB[CGSMini_Robot01LineBoxAnaInN01-EL3202]^RTD2^Status^Limit 1;
                        .stAnaRTDLine2.bTLimit2             := TIIB[CGSMini_Robot01LineBoxAnaInN01-EL3202]^RTD2^Status^Limit 2;
                        .stAnaRTDLine2.bTError              := TIIB[CGSMini_Robot01LineBoxAnaInN01-EL3202]^RTD2^Status^Error;
                        .stAnaRTDLine2.siAnaRaw             := TIIB[CGSMini_Robot01LineBoxAnaInN01-EL3202]^RTD2^Value;

                        .stAnaFlowLine1.bTUnderRange        := TIIB[CGSMini_Robot01LineBoxAnaInN02-EL3054]^Flow1^Status^Underrange;
                        .stAnaFlowLine1.bTOverRange         := TIIB[CGSMini_Robot01LineBoxAnaInN02-EL3054]^Flow1^Status^Overrange;
                        .stAnaFlowLine1.bTLimit1            := TIIB[CGSMini_Robot01LineBoxAnaInN02-EL3054]^Flow1^Status^Limit 1;
                        .stAnaFlowLine1.bTLimit2            := TIIB[CGSMini_Robot01LineBoxAnaInN02-EL3054]^Flow1^Status^Limit 2;
                        .stAnaFlowLine1.bTError             := TIIB[CGSMini_Robot01LineBoxAnaInN02-EL3054]^Flow1^Status^Error;
                        .stAnaFlowLine1.siAnaRaw            := TIIB[CGSMini_Robot01LineBoxAnaInN02-EL3054]^Flow1^Value;
                        
                        .stAnaFlowLine2.bTUnderRange        := TIIB[CGSMini_Robot01LineBoxAnaInN02-EL3054]^Flow2^Status^Underrange;
                        .stAnaFlowLine2.bTOverRange         := TIIB[CGSMini_Robot01LineBoxAnaInN02-EL3054]^Flow2^Status^Overrange;
                        .stAnaFlowLine2.bTLimit1            := TIIB[CGSMini_Robot01LineBoxAnaInN02-EL3054]^Flow2^Status^Limit 1;
                        .stAnaFlowLine2.bTLimit2            := TIIB[CGSMini_Robot01LineBoxAnaInN02-EL3054]^Flow2^Status^Limit 2;
                        .stAnaFlowLine2.bTError             := TIIB[CGSMini_Robot01LineBoxAnaInN02-EL3054]^Flow2^Status^Error;
                        .stAnaFlowLine2.siAnaRaw            := TIIB[CGSMini_Robot01LineBoxAnaInN02-EL3054]^Flow2^Value;
                       													
                        .stAnaPressure.bTUnderRange         := TIIB[CGSMini_Robot01LineBoxAnaInN02-EL3054]^Pressure1^Status^Underrange;
                        .stAnaPressure.bTOverRange          := TIIB[CGSMini_Robot01LineBoxAnaInN02-EL3054]^Pressure1^Status^Overrange;
                        .stAnaPressure.bTLimit1             := TIIB[CGSMini_Robot01LineBoxAnaInN02-EL3054]^Pressure1^Status^Limit 1;
                        .stAnaPressure.bTLimit2             := TIIB[CGSMini_Robot01LineBoxAnaInN02-EL3054]^Pressure1^Status^Limit 2;
                        .stAnaPressure.bTError              := TIIB[CGSMini_Robot01LineBoxAnaInN02-EL3054]^Pressure1^Status^Error;
                        .stAnaPressure.siAnaRaw             := TIIB[CGSMini_Robot01LineBoxAnaInN02-EL3054]^Pressure1^Value;

                        .stAnaRTDInternal.bTUnderRange      := TIIB[CGSMini_Robot01LineBoxAnaInN03-EL3202]^RTDInternal^Status^Underrange;
                        .stAnaRTDInternal.bTOverRange       := TIIB[CGSMini_Robot01LineBoxAnaInN03-EL3202]^RTDInternal^Status^Overrange;
                        .stAnaRTDInternal.bTLimit1          := TIIB[CGSMini_Robot01LineBoxAnaInN03-EL3202]^RTDInternal^Status^Limit 1;
                        .stAnaRTDInternal.bTLimit2          := TIIB[CGSMini_Robot01LineBoxAnaInN03-EL3202]^RTDInternal^Status^Limit 2;
                        .stAnaRTDInternal.bTError           := TIIB[CGSMini_Robot01LineBoxAnaInN03-EL3202]^RTDInternal^Status^Error;
                        .stAnaRTDInternal.siAnaRaw          := TIIB[CGSMini_Robot01LineBoxAnaInN03-EL3202]^RTDInternal^Value;

                        .stAnaRTDExternal.bTUnderRange      := TIIB[CGSMini_Robot01LineBoxAnaInN03-EL3202]^RTDExternal^Status^Underrange;
                        .stAnaRTDExternal.bTOverRange       := TIIB[CGSMini_Robot01LineBoxAnaInN03-EL3202]^RTDExternal^Status^Overrange;
                        .stAnaRTDExternal.bTLimit1          := TIIB[CGSMini_Robot01LineBoxAnaInN03-EL3202]^RTDExternal^Status^Limit 1;
                        .stAnaRTDExternal.bTLimit2          := TIIB[CGSMini_Robot01LineBoxAnaInN03-EL3202]^RTDExternal^Status^Limit 2;
                        .stAnaRTDExternal.bTError           := TIIB[CGSMini_Robot01LineBoxAnaInN03-EL3202]^RTDExternal^Status^Error;
                        .stAnaRTDExternal.siAnaRaw          := TIIB[CGSMini_Robot01LineBoxAnaInN03-EL3202]^RTDExternal^Value;
                        
                        .stOverCProt.bEnabled               := TIIB[CGSMini_Robot01LineBoxOverCurrProt1-EL9222]^OCP Inputs Channel 1^Status^Enabled;
                        .stOverCProt.bError                 := TIIB[CGSMini_Robot01LineBoxOverCurrProt1-EL9222]^OCP Inputs Channel 1^Status^Error;'}
  stBoxIN AT %I*:ST_RobotLineBox_HWI;

{attribute 'TcLinkTo':='.stOverCProtOut.bCtrlResetCh1       := TIIB[CGSMini_Robot01LineBoxOverCurrProt1-EL9222]^OCP Outputs Channel 1^Control^Reset;
                        .stOverCProtOut.bCtrlSwitchCh1      := TIIB[CGSMini_Robot01LineBoxOverCurrProt1-EL9222]^OCP Outputs Channel 1^Control^Switch;
                        .stOverCProtOut.bCtrlResetCh2       := TIIB[CGSMini_Robot01LineBoxOverCurrProt1-EL9222]^OCP Outputs Channel 2^Control^Reset;
                        .stOverCProtOut.bCtrlSwitchCh2      := TIIB[CGSMini_Robot01LineBoxOverCurrProt1-EL9222]^OCP Outputs Channel 2^Control^Switch;'}
  stBoxOUT AT %Q*:ST_RobotLineBox_HWQ;
  
{attribute 'TcLinkTo':='.stAnaInN04_3054State.uiDataState   := TIIB[CGSMini_Robot01OnBoardBoxAnaInN04-EL3054]^InfoData^State;
                        .stAnaInN04_3054State.bWCState      := TIIB[CGSMini_Robot01OnBoardBoxAnaInN04-EL3054]^WcState^WcState;
                        .stOnboardBox_1100State.uiDataState := TIIB[CGSMini_Robot01OnboardBox-EK1100]^InfoData^State;
                        .stOutN01_2008State.uiDataState     := TIIB[CGSMini_Robot01OnBoardBoxOutN01-EL2008]^InfoData^State;
                        .stOutN01_2008State.bWCState        := TIIB[CGSMini_Robot01OnBoardBoxOutN01-EL2008]^WcState^WcState;
                        
                        .stLaserPos_State.uiDataState       := TIIB[CGSMini_Robot01Laser-SickDL100]^InfoData^State;
                        .stLaserPos_State.bWCState          := TIIB[CGSMini_Robot01Laser-SickDL100]^WcState^WcState;
                        .stLaserPos.udiDistanceRaw          := TIIB[CGSMini_Robot01Laser-SickDL100]^Distance^Distance;
                        
                        .stAnaOnboardSpare1.bTUnderRange    := TIIB[CGSMini_Robot01OnBoardBoxAnaInN04-EL3054]^Spare1^Status^Underrange;
                        .stAnaOnboardSpare1.bTOverRange     := TIIB[CGSMini_Robot01OnBoardBoxAnaInN04-EL3054]^Spare1^Status^Overrange;
                        .stAnaOnboardSpare1.bTLimit1        := TIIB[CGSMini_Robot01OnBoardBoxAnaInN04-EL3054]^Spare1^Status^Limit 1;
                        .stAnaOnboardSpare1.bTLimit2        := TIIB[CGSMini_Robot01OnBoardBoxAnaInN04-EL3054]^Spare1^Status^Limit 2;
                        .stAnaOnboardSpare1.bTError         := TIIB[CGSMini_Robot01OnBoardBoxAnaInN04-EL3054]^Spare1^Status^Error;
                        .stAnaOnboardSpare1.siAnaRaw        := TIIB[CGSMini_Robot01OnBoardBoxAnaInN04-EL3054]^Spare1^Value;
  
                        .stPwrSupplyAX8620.comState.uiDataState:= TIIB[CGSMini_Robot01OnboardAxisPwrSupply-AX8620]^InfoData^State;
                        .stPwrSupplyAX8620.comState.bWcState   := TIIB[CGSMini_Robot01OnboardAxisPwrSupply-AX8620]^WcState^WcState;
                        .stPwrSupplyAX8620.sdiDcOutputShift := TIIB[CGSMini_Robot01OnboardAxisPwrSupply-AX8620]^InfoData^DcOutputShift;
                        .stPwrSupplyAX8620.sdiDcInputShift  := TIIB[CGSMini_Robot01OnboardAxisPwrSupply-AX8620]^InfoData^DcInputShift;
                        .stPwrSupplyAX8620.bOverTemp        := TIIB[CGSMini_Robot01OnboardAxisPwrSupply-AX8620]^PSM Warning register^Warning^A2 Device overtemperature;  
                        .stPwrSupplyAX8620.bFanMalfunc      := TIIB[CGSMini_Robot01OnboardAxisPwrSupply-AX8620]^PSM Warning register^Warning^A4 Fan malfunction;
                        .stPwrSupplyAX8620.bUnderVoltage    := TIIB[CGSMini_Robot01OnboardAxisPwrSupply-AX8620]^PSM Warning register^Warning^A6 Mains undervoltage;
                        .stPwrSupplyAX8620.bOverVoltage     := TIIB[CGSMini_Robot01OnboardAxisPwrSupply-AX8620]^PSM Warning register^Warning^A5 Mains overvoltage;
                        
                        .stDriverLine1.comState             := TIIB[CGSMini_Robot01OnboardAxisPwrSupply-AX8620]^CGSMini_Robot01OnboardAxisDriverLine1-AX8206^InfoData^State;
                        .stDriverLine1.sdiDcOutputShift     := TIIB[CGSMini_Robot01OnboardAxisPwrSupply-AX8620]^CGSMini_Robot01OnboardAxisDriverLine1-AX8206^InfoData^DcOutputShift;
                        .stDriverLine1.sdiDcInputShift      := TIIB[CGSMini_Robot01OnboardAxisPwrSupply-AX8620]^CGSMini_Robot01OnboardAxisDriverLine1-AX8206^InfoData^DcInputShift;                       
                        .stDriverLine1.siFrontIGBTTemp      := TIIB[CGSMini_Robot01OnboardAxisPwrSupply-AX8620]^CGSMini_Robot01OnboardAxisDriverLine1-AX8206^Front^Ch B AxisMain Inputs^IGBT temperature;
                        .stDriverLine1.udFrontMotorDIGIns   := TIIB[CGSMini_Robot01OnboardAxisPwrSupply-AX8620]^CGSMini_Robot01OnboardAxisDriverLine1-AX8206^Front^Ch B AxisMain Inputs^Ch B Digital inputs;                      
                        .stDriverLine1.siBackIGBTTemp       := TIIB[CGSMini_Robot01OnboardAxisPwrSupply-AX8620]^CGSMini_Robot01OnboardAxisDriverLine1-AX8206^Back^Ch A AxisMain Inputs^IGBT temperature;                                                
                        .stDriverLine1.udBackMotorDIGIns    := TIIB[CGSMini_Robot01OnboardAxisPwrSupply-AX8620]^CGSMini_Robot01OnboardAxisDriverLine1-AX8206^Back^Ch A AxisMain Inputs^Ch A Digital inputs;
                        .stDriverLine1.rFrontMotorTemp     := TIIB[CGSMini_Robot01OnboardAxisPwrSupply-AX8620]^CGSMini_Robot01OnboardAxisDriverLine1-AX8206^Front^Ch B SyncServoMotor Inputs^Actual motor temperature;
                        .stDriverLine1.rBackMotorTemp      := TIIB[CGSMini_Robot01OnboardAxisPwrSupply-AX8620]^CGSMini_Robot01OnboardAxisDriverLine1-AX8206^Back^Ch A SyncServoMotor Inputs^Actual motor temperature;                         
                        .stDriverLine1.rFrontMotorTorque    := TIIB[CGSMini_Robot01OnboardAxisPwrSupply-AX8620]^CGSMini_Robot01OnboardAxisDriverLine1-AX8206^Front^Ch B TorqueControl Inputs^Ch B Torque/force actual value;
                        .stDriverLine1.rBackMotorTorque     := TIIB[CGSMini_Robot01OnboardAxisPwrSupply-AX8620]^CGSMini_Robot01OnboardAxisDriverLine1-AX8206^Back^Ch A TorqueControl Inputs^Ch A Torque/force actual value;


                        .stDriverLine2.comState             := TIIB[CGSMini_Robot01OnboardAxisPwrSupply-AX8620]^CGSMini_Robot01OnboardAxisDriverLine2-AX8206^InfoData^State;
                        .stDriverLine2.sdiDcOutputShift     := TIIB[CGSMini_Robot01OnboardAxisPwrSupply-AX8620]^CGSMini_Robot01OnboardAxisDriverLine2-AX8206^InfoData^DcOutputShift;
                        .stDriverLine2.sdiDcInputShift      := TIIB[CGSMini_Robot01OnboardAxisPwrSupply-AX8620]^CGSMini_Robot01OnboardAxisDriverLine2-AX8206^InfoData^DcInputShift;                       
                        .stDriverLine2.siFrontIGBTTemp      := TIIB[CGSMini_Robot01OnboardAxisPwrSupply-AX8620]^CGSMini_Robot01OnboardAxisDriverLine2-AX8206^Front^Ch B AxisMain Inputs^IGBT temperature;
                        .stDriverLine2.udFrontMotorDIGIns   := TIIB[CGSMini_Robot01OnboardAxisPwrSupply-AX8620]^CGSMini_Robot01OnboardAxisDriverLine2-AX8206^Front^Ch B AxisMain Inputs^Ch B Digital inputs;                       
                        .stDriverLine2.siBackIGBTTemp       := TIIB[CGSMini_Robot01OnboardAxisPwrSupply-AX8620]^CGSMini_Robot01OnboardAxisDriverLine2-AX8206^Back^Ch A AxisMain Inputs^IGBT temperature;
                        .stDriverLine2.udBackMotorDIGIns    := TIIB[CGSMini_Robot01OnboardAxisPwrSupply-AX8620]^CGSMini_Robot01OnboardAxisDriverLine2-AX8206^Back^Ch A AxisMain Inputs^Ch A Digital inputs;                        
                        .stDriverLine2.rFrontMotorTemp      := TIIB[CGSMini_Robot01OnboardAxisPwrSupply-AX8620]^CGSMini_Robot01OnboardAxisDriverLine2-AX8206^Front^Ch B SyncServoMotor Inputs^Actual motor temperature;
                        .stDriverLine2.rBackMotorTemp       := TIIB[CGSMini_Robot01OnboardAxisPwrSupply-AX8620]^CGSMini_Robot01OnboardAxisDriverLine2-AX8206^Back^Ch A SyncServoMotor Inputs^Actual motor temperature;                       
                        .stDriverLine2.rFrontMotorTorque    := TIIB[CGSMini_Robot01OnboardAxisPwrSupply-AX8620]^CGSMini_Robot01OnboardAxisDriverLine2-AX8206^Front^Ch B TorqueControl Inputs^Ch B Torque/force actual value;
                        .stDriverLine2.rBackMotorTorque     := TIIB[CGSMini_Robot01OnboardAxisPwrSupply-AX8620]^CGSMini_Robot01OnboardAxisDriverLine2-AX8206^Back^Ch A TorqueControl Inputs^Ch A Torque/force actual value;'}
  stIN AT %I*:ST_Robot_HWI;


{attribute 'TcLinkTo':='.FlushFloor                          := TIIB[CGSMini_Robot01OnBoardBoxOutN01-EL2008]^Channel 1^FlushFloor;
                        .IrrigLine1                          := TIIB[CGSMini_Robot01OnBoardBoxOutN01-EL2008]^Channel 3^IrrigLine1;
                        .IrrigLine2                          := TIIB[CGSMini_Robot01OnBoardBoxOutN01-EL2008]^Channel 4^IrrigLine2;'}
  stOUT AT %Q*:ST_Robot_HWQ;

{attribute 'TcNcAxis' := '.Line1Front                       := CGSMini_Robot01AxisLine1Front;
                          .Line1Back                        := CGSMini_Robot01AxisLine1Back;
                          .Line2Front                       := CGSMini_Robot01AxisLine2Front;
                          .Line2Back                        := CGSMini_Robot01AxisLine2Back;'}
  stAxes : ST_Robot_Axes;
  
END_VAR

// ---- GVLs/GQ.TcGVL
{attribute 'qualified_only'}
{IF defined (debugCompile)}
//contains ONLY global variable to access hardware output debugCompile mode
{info '---------------simulation output global variables used; DEBUG defined---------------'}
VAR_GLOBAL
  //contains ONLY global variable for outputs
  stMainCabinet 				: ST_MainCabinet_HWQ;	
END_VAR
{END_IF}


VAR_GLOBAL
  {info '---------------Hardware outputs used; CGSMiniRobot defined---------------'}
  {attribute 'TcLinkTo':='.bEmgyBtnWhiteLight     := TIIB[CGSMini_RobotAllMainCabOutN01-EL2008]^Channel 2^EmgyBtnWhiteLight;
                          .bEmgyBtnRedLight       := TIIB[CGSMini_RobotAllMainCabOutN01-EL2008]^Channel 3^EmgyBtnRedLight;
                          
                          .stStackLight.bBlue		  := TIIB[CGSMini_RobotAllMainCabOutN01-EL2008]^Channel 4^blue;
                          .stStackLight.bGreen    := TIIB[CGSMini_RobotAllMainCabOutN01-EL2008]^Channel 5^green;
                          .stStackLight.bOrange   := TIIB[CGSMini_RobotAllMainCabOutN01-EL2008]^Channel 6^orange;
                          .stStackLight.bRed      := TIIB[CGSMini_RobotAllMainCabOutN01-EL2008]^Channel 7^red;
                          .stStackLight.bBuzzer	  := TIIB[CGSMini_RobotAllMainCabOutN01-EL2008]^Channel 8^buzzer;'}
  stMainCabinet AT %Q* :ST_MainCabinet_HWQ;	
END_VAR

// ---- POUs/MAIN.TcPOU
PROGRAM MAIN
VAR
   i : INT;
END_VAR

i := i + 1;

END_PROGRAM
